(* IEC 61131-3 sources: 2026_Projet_YGO_ExcavatriceDragage/TOOLS/TEST_AUTO_CI/RESULTS/_TROUBLESHOOTING/tests, 5 files *)

(* ---- test_arb_cmd_both_atomic.st ---- *)
(* =========================================================================
   TEST CI AD HOC - Atomicite commande Both M1/M2 (T216, criticite C4)
   -------------------------------------------------------------------------
   Prouve les invariants de securite du depart couple des treuils M1/M2 :
     #1  Atomicite Both descente : BothDescendPermit=FALSE (un permit M2 absent)
         -> AUCUN des deux treuils ne demarre (StartStop M1=FALSE ET M2=FALSE).
     #2  Both nominal montee : les 2 permits agreges OK -> les DEUX demarrent.
     #3  Preservation unitaire : M1 seul / M2 seul / action benne M2 -> le gate
         Both*Permit est inactif, comportement inchange (aucun blocage croise).
     #4  Soft-stop : Both + ecart mineur -> jamais de demarrage unilateral (les 2
         bloques ensemble si le permit Both manque) ; hors Both (unitaire), l'ecart
         mineur bloque toujours le sens concerne (comportement preserve).
   Noms figes T216 intacts : EffectivePermitM1/2_Ascent/Descend non re-nommes.
   Chaque appel arb1(...)/arb2(...) = 1 scan de l'arbitre.
   (Le gate sync mineur de PRG_04 est coupe en Both en amont - voir le FB - ici on
   prouve que l'arbitre ne part JAMAIS seul, quelle que soit la polarite du flag.)
   ========================================================================= *)

SETUP
VAR
    arb1 : FB_WinchCmdArbitrationM1;
    arb2 : FB_WinchCmdArbitrationM2;
    joy  : ST_AcquisitionJoystickQualified;
    auth : ST_Modes_Autorisations;
    req  : ST_ProgramWinchRequest;
    both : ST_WinchBothIntent;
    ihm  : ST_fbWinchCmdArbitration_IHM;
    ctx  : ST_fbWinchCmdArbitration_Context;
    cfg1 : ST_fbWinchCmdArbitration_Cfg;
    cfg2 : ST_fbWinchCmdArbitration_Cfg;
END_VAR
END_SETUP

TEST 'T216 #1 Atomicite Both descente : BothDescendPermit=FALSE -> AUCUN treuil ne demarre'
    // Contexte : mode manuel boutons, intention both descente active.
    auth.Mode := E_Mode.MAINT_N1;
    auth.JoystickWinchSelectArbitrated := 0;
    both.Active := TRUE; both.Direction := -1;
    // Simule EffectivePermitM2_Descend=FALSE -> BothDescendPermit=FALSE (agregat PRG_04).
    ctx.BothDescendPermit := FALSE; ctx.BothAscentPermit := TRUE;
    ctx.BothBlock := TRUE;
    ctx.BucketBusy := FALSE; ctx.WinchBothMotionBlockedByBucket := FALSE;
    ctx.SyncBlocksAscent := FALSE; ctx.SyncBlocksDescent := FALSE;
    ihm.BtnAscentM1 := FALSE; ihm.BtnDescentM1 := FALSE;
    ihm.BtnAscentM2 := FALSE; ihm.BtnDescentM2 := FALSE;
    cfg1.BtnStepTgt := 5; cfg2.BtnStepTgt := 5; cfg2.BucketOverrideStepTgt := 1;

    arb1(Enable := TRUE, Joystick := joy, Auth := auth, ReqWinch := req,
         BothIntent := both, IHM := ihm, TglJoystickMaster := FALSE,
         Context := ctx, Cfg := cfg1);
    arb2(Enable := TRUE, Joystick := joy, Auth := auth, ReqWinch := req,
         BothIntent := both, IHM := ihm, TglJoystickMaster := FALSE,
         Context := ctx, Cfg := cfg2);

    ASSERT_FALSE(arb1.StartStop, 'T216#1 Both descente : StartStop M1=FALSE (permit Both manquant)');
    ASSERT_FALSE(arb2.StartStop, 'T216#1 Both descente : StartStop M2=FALSE (permit Both manquant)');
    ASSERT_EQ(arb1.Direction, -1, 'T216#1 l intention descente est portee, seule la commande est coupee');
END_TEST

TEST 'T216 #2 Both nomiinal montee : permits OK -> les DEUX demarrent ensemble'
    auth.Mode := E_Mode.MAINT_N1;
    auth.JoystickWinchSelectArbitrated := 0;
    both.Active := TRUE; both.Direction := 1;
    ctx.BothDescendPermit := TRUE; ctx.BothAscentPermit := TRUE;
    ctx.BothBlock := FALSE;
    ctx.BucketBusy := FALSE; ctx.WinchBothMotionBlockedByBucket := FALSE;
    ctx.SyncBlocksAscent := FALSE; ctx.SyncBlocksDescent := FALSE;
    ihm.BtnAscentM1 := FALSE; ihm.BtnDescentM1 := FALSE;
    ihm.BtnAscentM2 := FALSE; ihm.BtnDescentM2 := FALSE;
    cfg1.BtnStepTgt := 5; cfg2.BtnStepTgt := 5; cfg2.BucketOverrideStepTgt := 1;

    arb1(Enable := TRUE, Joystick := joy, Auth := auth, ReqWinch := req,
         BothIntent := both, IHM := ihm, TglJoystickMaster := FALSE,
         Context := ctx, Cfg := cfg1);
    arb2(Enable := TRUE, Joystick := joy, Auth := auth, ReqWinch := req,
         BothIntent := both, IHM := ihm, TglJoystickMaster := FALSE,
         Context := ctx, Cfg := cfg2);

    ASSERT_TRUE(arb1.StartStop, 'T216#2 Both montee : M1 demarre (permit OK)');
    ASSERT_TRUE(arb2.StartStop, 'T216#2 Both montee : M2 demarre (permit OK)');
    ASSERT_EQ(arb1.Direction, 1, 'T216#2 M1 sens montee');
    ASSERT_EQ(arb2.Direction, 1, 'T216#2 M2 sens montee');
END_TEST

TEST 'T216 #3a M1 seul : gate Both inactif (pas de blocage croise)'
    auth.Mode := E_Mode.MAINT_N1;
    auth.JoystickWinchSelectArbitrated := 1;
    both.Active := FALSE; both.Direction := 0;
    // Meme si les permits Both sont faux, le pilotage unitaire M1 n'en depend pas.
    ctx.BothDescendPermit := FALSE; ctx.BothAscentPermit := FALSE;
    ctx.BothBlock := FALSE;
    ctx.BucketBusy := FALSE; ctx.WinchBothMotionBlockedByBucket := FALSE;
    ctx.SyncBlocksAscent := FALSE; ctx.SyncBlocksDescent := FALSE;
    ihm.BtnAscentM1 := TRUE; ihm.BtnDescentM1 := FALSE;
    cfg1.BtnStepTgt := 5; cfg2.BtnStepTgt := 5; cfg2.BucketOverrideStepTgt := 1;

    arb1(Enable := TRUE, Joystick := joy, Auth := auth, ReqWinch := req,
         BothIntent := both, IHM := ihm, TglJoystickMaster := FALSE,
         Context := ctx, Cfg := cfg1);

    ASSERT_TRUE(arb1.StartStop, 'T216#3a M1 seul : demarre (couplage Both inactif)');
    ASSERT_EQ(arb1.Direction, 1, 'T216#3a M1 sens montee');
END_TEST

TEST 'T216 #3b M2 seul : gate Both inactif (pas de blocage croise)'
    auth.Mode := E_Mode.MAINT_N1;
    auth.JoystickWinchSelectArbitrated := 2;
    both.Active := FALSE; both.Direction := 0;
    ctx.BothDescendPermit := FALSE; ctx.BothAscentPermit := FALSE;
    ctx.BothBlock := FALSE;
    ctx.BucketBusy := FALSE; ctx.WinchBothMotionBlockedByBucket := FALSE;
    ctx.SyncBlocksAscent := FALSE; ctx.SyncBlocksDescent := FALSE;
    ihm.BtnAscentM2 := TRUE;

    arb2(Enable := TRUE, Joystick := joy, Auth := auth, ReqWinch := req,
         BothIntent := both, IHM := ihm, TglJoystickMaster := FALSE,
         Context := ctx, Cfg := cfg2);

    ASSERT_TRUE(arb2.StartStop, 'T216#3b M2 seul : demarre (couplage Both inactif)');
    ASSERT_EQ(arb2.Direction, 1, 'T216#3b M2 sens montee');
END_TEST

TEST 'T216 #3c benne M2 : chemin override preserve (hors gate Both)'
    auth.Mode := E_Mode.MAINT_N1;
    both.Active := FALSE; both.Direction := 0;
    ctx.BothDescendPermit := FALSE; ctx.BothAscentPermit := FALSE;
    ctx.BothBlock := FALSE;
    // Action benne M2 active (chemin override FB_WinchCmdArbitrationM2).
    ctx.BucketBusy := TRUE; ctx.BucketM2StartStop := TRUE; ctx.BucketM2Open := TRUE;
    ctx.WinchBothMotionBlockedByBucket := FALSE;
    ctx.SyncBlocksAscent := FALSE; ctx.SyncBlocksDescent := FALSE;
    cfg2.BucketOverrideStepTgt := 1;

    arb2(Enable := TRUE, Joystick := joy, Auth := auth, ReqWinch := req,
         BothIntent := both, IHM := ihm, TglJoystickMaster := FALSE,
         Context := ctx, Cfg := cfg2);

    ASSERT_TRUE(arb2.StartStop, 'T216#3c action benne M2 : demarre (override hors gate Both)');
    ASSERT_EQ(arb2.StepTgt, 1, 'T216#3c action benne M2 : palier lent override');
END_TEST

TEST 'T216 #4a Both + ecart mineur : JAMAIS de demarrage unilateral (les DEUX bloques)'
    auth.Mode := E_Mode.MAINT_N1;
    auth.JoystickWinchSelectArbitrated := 0;
    both.Active := TRUE; both.Direction := -1;
    ctx.BothDescendPermit := FALSE;   // un permit Both manquant (M2)
    ctx.BothAscentPermit := TRUE;
    ctx.BothBlock := TRUE;
    ctx.BucketBusy := FALSE; ctx.WinchBothMotionBlockedByBucket := FALSE;
    // M1 bloque sur SyncBlocksAscent ; en descente M2 bloque sur SyncBlocksDescent.
    // Quelle que soit la polarite, le gate Both (permit manquant) bloque les DEUX.
    ctx.SyncBlocksAscent := TRUE; ctx.SyncBlocksDescent := TRUE;

    arb1(Enable := TRUE, Joystick := joy, Auth := auth, ReqWinch := req,
         BothIntent := both, IHM := ihm, TglJoystickMaster := FALSE,
         Context := ctx, Cfg := cfg1);
    arb2(Enable := TRUE, Joystick := joy, Auth := auth, ReqWinch := req,
         BothIntent := both, IHM := ihm, TglJoystickMaster := FALSE,
         Context := ctx, Cfg := cfg2);

    ASSERT_FALSE(arb1.StartStop, 'T216#4a Both + ecart : M1 bloque (pas de depart unilateral)');
    ASSERT_FALSE(arb2.StartStop, 'T216#4a Both + ecart : M2 bloque (pas de depart unilateral)');
END_TEST

TEST 'T216 #4b unite + ecart mineur : le sens concerne reste bloque (preservation)'
    auth.Mode := E_Mode.MAINT_N1;
    auth.JoystickWinchSelectArbitrated := 1;
    both.Active := FALSE; both.Direction := 0;
    ctx.BothDescendPermit := FALSE; ctx.BothAscentPermit := FALSE;
    ctx.BothBlock := FALSE;
    ctx.BucketBusy := FALSE; ctx.WinchBothMotionBlockedByBucket := FALSE;
    // Montee M1 bloquee par l'ecart mineur si SyncBlocksAscent (comportement d'origine
    // hors Both, preserve).
    ctx.SyncBlocksAscent := TRUE; ctx.SyncBlocksDescent := FALSE;
    ihm.BtnAscentM1 := TRUE;

    arb1(Enable := TRUE, Joystick := joy, Auth := auth, ReqWinch := req,
         BothIntent := both, IHM := ihm, TglJoystickMaster := FALSE,
         Context := ctx, Cfg := cfg1);

    ASSERT_FALSE(arb1.StartStop, 'T216#4b M1 seul + ecart mineur montee : bloque (comportement preserve hors Both)');
END_TEST

(* ---- test_fb_encoder_speedmeasure.st ---- *)
SETUP
VAR
    fb : FB_Encoder_SpeedMeasure;
END_VAR
END_SETUP

TEST 'TC-T084-001 Mesure dynamique 1.0 m/s et 2.0 m/s sur fenetre glissante 50ms'
    (* Scan 0 : Neutralisation initiale *)
    fb(Enable := FALSE, Reset := FALSE, Position_M := 0.0, PositionValid := FALSE);
    ASSERT_FALSE(fb.Valid, 'Enable=FALSE -> Valid=FALSE');
    ASSERT_EQ(fb.Speed_Mps, 0.0, 'Enable=FALSE -> Speed=0');

    ADVANCE_TIME(10000000); (* +10 ms *)

    (* Scan 1 (t=10ms) : Activation et premier echantillon a 0.0 m *)
    fb(Enable := TRUE, Reset := FALSE, Position_M := 0.0, PositionValid := TRUE);
    ASSERT_FALSE(fb.Valid, 'Echantillon 1 : Fenetre 50ms pas encore remplie');

    ADVANCE_TIME(10000000); (* +10 ms (t=20ms) *)

    (* Scan 2 (t=20ms) : Deplacement a v=1.0 m/s -> pos = 0.01 m (+10mm en 10ms) *)
    fb(Enable := TRUE, Reset := FALSE, Position_M := 0.01, PositionValid := TRUE);
    ASSERT_FALSE(fb.Valid, 'Echantillon 2 : Fenetre 50ms pas encore remplie');

    ADVANCE_TIME(10000000); (* +10 ms (t=30ms) *)

    (* Scan 3 (t=30ms) : pos = 0.02 m *)
    fb(Enable := TRUE, Reset := FALSE, Position_M := 0.02, PositionValid := TRUE);
    ASSERT_FALSE(fb.Valid, 'Echantillon 3 : Fenetre 50ms pas encore remplie');

    ADVANCE_TIME(10000000); (* +10 ms (t=40ms) *)

    (* Scan 4 (t=40ms) : pos = 0.03 m *)
    fb(Enable := TRUE, Reset := FALSE, Position_M := 0.03, PositionValid := TRUE);
    ASSERT_FALSE(fb.Valid, 'Echantillon 4 : Fenetre 50ms pas encore remplie');

    ADVANCE_TIME(10000000); (* +10 ms (t=50ms) *)

    (* Scan 5 (t=50ms) : pos = 0.04 m *)
    fb(Enable := TRUE, Reset := FALSE, Position_M := 0.04, PositionValid := TRUE);
    ASSERT_FALSE(fb.Valid, 'Echantillon 5 : Fenetre 50ms pas encore remplie');

    ADVANCE_TIME(10000000); (* +10 ms (t=60ms) *)

    (* Scan 6 (t=60ms) : pos = 0.05 m -> 6 echantillons couvrant 50ms (t=10ms a t=60ms) *)
    fb(Enable := TRUE, Reset := FALSE, Position_M := 0.05, PositionValid := TRUE);
    ASSERT_TRUE(fb.Valid, '6 echantillons sur 50ms atteints -> Valid=TRUE');
    ASSERT_NEAR(fb.Speed_Mps, 1.0, 0.05, 'Vitesse absolue mesuree = 1.0 m/s');
    ASSERT_NEAR(fb.SignedSpeed_Mps, 1.0, 0.05, 'Vitesse signee montee = +1.0 m/s');

    ADVANCE_TIME(10000000); (* +10 ms (t=70ms) *)

    (* Scan 7 (t=70ms) : Acceleration a 2.0 m/s (+20mm en 10ms) -> pos = 0.07 m *)
    fb(Enable := TRUE, Reset := FALSE, Position_M := 0.07, PositionValid := TRUE);
    ASSERT_TRUE(fb.Valid, 'Fenetre glissante active');
    ASSERT_NEAR(fb.Speed_Mps, 1.2, 0.05, 'Transition glissante vers 2.0 m/s (pos 0.07 - pos 0.01 = 0.06m / 50ms = 1.2 m/s)');

    ADVANCE_TIME(10000000); (* +10 ms (t=80ms) *)

    (* Scan 8 (t=80ms) : Suite a 2.0 m/s -> pos = 0.09 m *)
    fb(Enable := TRUE, Reset := FALSE, Position_M := 0.09, PositionValid := TRUE);
    ASSERT_TRUE(fb.Valid, 'Fenetre glissante active');
    ASSERT_NEAR(fb.Speed_Mps, 1.4, 0.05, 'Transition glissante vers 2.0 m/s (pos 0.09 - pos 0.02 = 0.07m / 50ms = 1.4 m/s)');

    ADVANCE_TIME(10000000); (* +10 ms (t=90ms) *)

    (* Scan 9 (t=90ms) : Descente a -2.0 m/s (-20mm en 10ms) -> pos = 0.07 m *)
    fb(Enable := TRUE, Reset := FALSE, Position_M := 0.07, PositionValid := TRUE);
    ASSERT_TRUE(fb.Valid, 'Fenetre glissante active');

    ADVANCE_TIME(10000000); (* +10 ms (t=100ms) *)

    (* Scan 10 (t=100ms) : Coupure PositionValid=FALSE -> Purge immediate *)
    fb(Enable := TRUE, Reset := FALSE, Position_M := 0.07, PositionValid := FALSE);
    ASSERT_FALSE(fb.Valid, 'Rupture confiance PositionValid=FALSE -> Valid retombe immediatement a FALSE');
    ASSERT_EQ(fb.Speed_Mps, 0.0, 'Purge immediate -> Speed=0.0');
    ASSERT_EQ(fb.SignedSpeed_Mps, 0.0, 'Purge immediate -> SignedSpeed=0.0');
END_TEST

(* ---- test_fb_sim_joystick.st ---- *)
(* ═══════════════════════════════════════════════════════════════════════
   🕵️ TEST CI AD HOC — FB_Joystick / ArmingPermit (LOT_JOYSTICK_ARMINGPERMIT)
   ───────────────────────────────────────────────────────────────────────
   Prouve les critères d'acceptation AC1/AC2/AC3 du contrat
   TASK_CONTRACT_JOYSTICK_ARMINGPERMIT.yaml :
     • AC1 : ArmingPermit=FALSE + appui 110ms -> DeadmanArmed=FALSE ;
             ArmingPermit=TRUE  + appui 110ms -> DeadmanArmed=TRUE.
     • AC2 : ArmingPermit=FALSE -> AxisCmdX/Y.Enable=FALSE, SpeedRef=0,
             warning "armement non permis" actif (sortie ArmingPermitDenied).
     • AC3 : RawOutOfRange=TRUE -> Enable=FALSE même si ArmingPermit=TRUE ;
             ArmingPermit=FALSE bloque l'armement même sans défaut capteur.
   ⚠️ Chaque appel fb(...) = 1 scan (10ms) ; ADVANCE_TIME avance le temps simulé
   sans faire tourner le FB. Un maintien de 110ms = front + ADVANCE_TIME + rappel.
   ⚠️ STruCpp ne re-copie PAS la sortie VAR_IN_OUT (NeutralXMem/YMem) entre deux
   appels -> nx/ny ré-injectés avant chaque appel (limite outillage documentée).
   Chaque TEST remet l'état armement à zéro via un premier appel ENABLE:=FALSE
   (le gate remet DeadmanArmed/DeadmanArmPending/ArmingPermitDenied/timers) pour
   être autonome quelle que soit l'instance FB.
   ═══════════════════════════════════════════════════════════════════════ *)

SETUP
VAR
    fb : FB_JOYSTICK;
    nx : INT := 5000;
    ny : INT := 5000;
    diagOk : ST_DIAG_DEVICE;
END_VAR
END_SETUP

TEST 'AC1a : ArmingPermit=FALSE bloque l armement (appui maintenu 110ms)'
    diagOk.ONLINE := TRUE; diagOk.OPERATIONAL := TRUE; diagOk.ERROR := FALSE;
    diagOk.ERRORID := 0; diagOk.STATE := E_DIAG_STATE.READY; diagOk.STATEATERROR := E_DIAG_STATE.DISABLED;
    nx := 5000; ny := 5000;

    (* reset etat armement via le gate Enable=FALSE *)
    fb(ENABLE := FALSE, RESET := FALSE,
       ARMINGPERMIT := FALSE,
       BUSCANOPENOP := diagOk, JOYSTICKOP := diagOk,
       RAWX := 5000, RAWY := 5000, RAWBUTTON := FALSE, BTNCALIBRATE := FALSE,
       INVERTX := FALSE, INVERTY := FALSE, DEADBANDRAW := 300,
       NEUTRALHOLDTIME := T#100MS, DEADMANARMHOLDTIME := T#100MS, DEADMANARMGRACETIME := T#3S,
       NEUTRALXMEM := nx, NEUTRALYMEM := ny);

    (* front appui, ArmingPermit=FALSE : la permission refuse le démarrage du timer
       d'armement -> DeadmanArmed ne doit JAMAIS passer à TRUE. *)
    fb(ENABLE := TRUE, RESET := FALSE,
       ARMINGPERMIT := FALSE,
       BUSCANOPENOP := diagOk, JOYSTICKOP := diagOk,
       RAWX := 5000, RAWY := 5000, RAWBUTTON := TRUE, BTNCALIBRATE := FALSE,
       INVERTX := FALSE, INVERTY := FALSE, DEADBANDRAW := 300,
       NEUTRALHOLDTIME := T#100MS, DEADMANARMHOLDTIME := T#100MS, DEADMANARMGRACETIME := T#3S,
       NEUTRALXMEM := nx, NEUTRALYMEM := ny);
    ADVANCE_TIME(110000000);   (* maintien 110ms >= DeadmanArmHoldTime 100ms *)
    fb(ENABLE := TRUE, RESET := FALSE,
       ARMINGPERMIT := FALSE,
       BUSCANOPENOP := diagOk, JOYSTICKOP := diagOk,
       RAWX := 5000, RAWY := 5000, RAWBUTTON := TRUE, BTNCALIBRATE := FALSE,
       INVERTX := FALSE, INVERTY := FALSE, DEADBANDRAW := 300,
       NEUTRALHOLDTIME := T#100MS, DEADMANARMHOLDTIME := T#100MS, DEADMANARMGRACETIME := T#3S,
       NEUTRALXMEM := nx, NEUTRALYMEM := ny);
    ASSERT_FALSE(fb.DEADMANARMED, 'AC1 : ArmingPermit=FALSE + appui 110ms -> DeadmanArmed reste FALSE (armement bloque)');
END_TEST

TEST 'AC1b : ArmingPermit=TRUE autorise l armement (appui maintenu 110ms)'
    diagOk.ONLINE := TRUE; diagOk.OPERATIONAL := TRUE; diagOk.ERROR := FALSE;
    diagOk.ERRORID := 0; diagOk.STATE := E_DIAG_STATE.READY; diagOk.STATEATERROR := E_DIAG_STATE.DISABLED;
    nx := 5000; ny := 5000;

    fb(ENABLE := FALSE, RESET := FALSE,
       ARMINGPERMIT := TRUE,
       BUSCANOPENOP := diagOk, JOYSTICKOP := diagOk,
       RAWX := 5000, RAWY := 5000, RAWBUTTON := FALSE, BTNCALIBRATE := FALSE,
       INVERTX := FALSE, INVERTY := FALSE, DEADBANDRAW := 300,
       NEUTRALHOLDTIME := T#100MS, DEADMANARMHOLDTIME := T#100MS, DEADMANARMGRACETIME := T#3S,
       NEUTRALXMEM := nx, NEUTRALYMEM := ny);

    (* front appui, ArmingPermit=TRUE : maintien complet -> armement normal *)
    fb(ENABLE := TRUE, RESET := FALSE,
       ARMINGPERMIT := TRUE,
       BUSCANOPENOP := diagOk, JOYSTICKOP := diagOk,
       RAWX := 5000, RAWY := 5000, RAWBUTTON := TRUE, BTNCALIBRATE := FALSE,
       INVERTX := FALSE, INVERTY := FALSE, DEADBANDRAW := 300,
       NEUTRALHOLDTIME := T#100MS, DEADMANARMHOLDTIME := T#100MS, DEADMANARMGRACETIME := T#3S,
       NEUTRALXMEM := nx, NEUTRALYMEM := ny);
    ADVANCE_TIME(110000000);   (* maintien 110ms >= DeadmanArmHoldTime 100ms *)
    fb(ENABLE := TRUE, RESET := FALSE,
       ARMINGPERMIT := TRUE,
       BUSCANOPENOP := diagOk, JOYSTICKOP := diagOk,
       RAWX := 5000, RAWY := 5000, RAWBUTTON := TRUE, BTNCALIBRATE := FALSE,
       INVERTX := FALSE, INVERTY := FALSE, DEADBANDRAW := 300,
       NEUTRALHOLDTIME := T#100MS, DEADMANARMHOLDTIME := T#100MS, DEADMANARMGRACETIME := T#3S,
       NEUTRALXMEM := nx, NEUTRALYMEM := ny);
    ASSERT_TRUE(fb.DEADMANARMED, 'AC1 : ArmingPermit=TRUE + appui 110ms -> DeadmanArmed=TRUE (armement autorise)');
END_TEST

TEST 'AC2 : ArmingPermit=FALSE -> Enable=FALSE, SpeedRef=0, warning armement non permis actif'
    diagOk.ONLINE := TRUE; diagOk.OPERATIONAL := TRUE; diagOk.ERROR := FALSE;
    diagOk.ERRORID := 0; diagOk.STATE := E_DIAG_STATE.READY; diagOk.STATEATERROR := E_DIAG_STATE.DISABLED;
    nx := 5000; ny := 5000;

    fb(ENABLE := FALSE, RESET := FALSE,
       ARMINGPERMIT := FALSE,
       BUSCANOPENOP := diagOk, JOYSTICKOP := diagOk,
       RAWX := 5000, RAWY := 5000, RAWBUTTON := FALSE, BTNCALIBRATE := FALSE,
       INVERTX := FALSE, INVERTY := FALSE, DEADBANDRAW := 300,
       NEUTRALHOLDTIME := T#100MS, DEADMANARMHOLDTIME := T#100MS, DEADMANARMGRACETIME := T#3S,
       NEUTRALXMEM := nx, NEUTRALYMEM := ny);

    (* appui maintenu, ArmingPermit=FALSE : armement bloqué. On pousse même l'axe X/Y
       (RawX/Y=8000) pour prouver qu'AUCUNE commande de mouvement n'est émise. *)
    fb(ENABLE := TRUE, RESET := FALSE,
       ARMINGPERMIT := FALSE,
       BUSCANOPENOP := diagOk, JOYSTICKOP := diagOk,
       RAWX := 5000, RAWY := 5000, RAWBUTTON := TRUE, BTNCALIBRATE := FALSE,
       INVERTX := FALSE, INVERTY := FALSE, DEADBANDRAW := 300,
       NEUTRALHOLDTIME := T#100MS, DEADMANARMHOLDTIME := T#100MS, DEADMANARMGRACETIME := T#3S,
       NEUTRALXMEM := nx, NEUTRALYMEM := ny);
    ADVANCE_TIME(110000000);
    fb(ENABLE := TRUE, RESET := FALSE,
       ARMINGPERMIT := FALSE,
       BUSCANOPENOP := diagOk, JOYSTICKOP := diagOk,
       RAWX := 8000, RAWY := 8000, RAWBUTTON := TRUE, BTNCALIBRATE := FALSE,
       INVERTX := FALSE, INVERTY := FALSE, DEADBANDRAW := 300,
       NEUTRALHOLDTIME := T#100MS, DEADMANARMHOLDTIME := T#100MS, DEADMANARMGRACETIME := T#3S,
       NEUTRALXMEM := nx, NEUTRALYMEM := ny);
    ASSERT_FALSE(fb.DEADMANARMED, 'AC2 : pre-requis - armement bloque (jamais arme)');
    ASSERT_FALSE(fb.AXISCMDX.ENABLE, 'AC2 : ArmingPermit=FALSE -> AxisCmdX.Enable=FALSE (pipeline neutralise)');
    ASSERT_FALSE(fb.AXISCMDY.ENABLE, 'AC2 : ArmingPermit=FALSE -> AxisCmdY.Enable=FALSE');
    ASSERT_NEAR(fb.AXISCMDX.SPEEDREF, 0.0, 0.01, 'AC2 : SpeedRef axe X = 0 (aucune commande de mouvement)');
    ASSERT_NEAR(fb.AXISCMDY.SPEEDREF, 0.0, 0.01, 'AC2 : SpeedRef axe Y = 0');
    ASSERT_TRUE(fb.ARMINGPERMITDENIED, 'AC2 : warning "armement non permis" actif (sortie dediee ArmingPermitDenied)');
END_TEST

TEST 'AC3a : defaut capteur (RawOutOfRange) neutralise Enable meme si ArmingPermit=TRUE'
    diagOk.ONLINE := TRUE; diagOk.OPERATIONAL := TRUE; diagOk.ERROR := FALSE;
    diagOk.ERRORID := 0; diagOk.STATE := E_DIAG_STATE.READY; diagOk.STATEATERROR := E_DIAG_STATE.DISABLED;
    nx := 5000; ny := 5000;

    fb(ENABLE := FALSE, RESET := FALSE,
       ARMINGPERMIT := TRUE,
       BUSCANOPENOP := diagOk, JOYSTICKOP := diagOk,
       RAWX := 5000, RAWY := 5000, RAWBUTTON := FALSE, BTNCALIBRATE := FALSE,
       INVERTX := FALSE, INVERTY := FALSE, DEADBANDRAW := 300,
       NEUTRALHOLDTIME := T#100MS, DEADMANARMHOLDTIME := T#100MS, DEADMANARMGRACETIME := T#3S,
       NEUTRALXMEM := nx, NEUTRALYMEM := ny);

    (* arme d'abord avec ArmingPermit=TRUE *)
    fb(ENABLE := TRUE, RESET := FALSE,
       ARMINGPERMIT := TRUE,
       BUSCANOPENOP := diagOk, JOYSTICKOP := diagOk,
       RAWX := 5000, RAWY := 5000, RAWBUTTON := TRUE, BTNCALIBRATE := FALSE,
       INVERTX := FALSE, INVERTY := FALSE, DEADBANDRAW := 300,
       NEUTRALHOLDTIME := T#100MS, DEADMANARMHOLDTIME := T#100MS, DEADMANARMGRACETIME := T#3S,
       NEUTRALXMEM := nx, NEUTRALYMEM := ny);
    ADVANCE_TIME(110000000);
    fb(ENABLE := TRUE, RESET := FALSE,
       ARMINGPERMIT := TRUE,
       BUSCANOPENOP := diagOk, JOYSTICKOP := diagOk,
       RAWX := 5000, RAWY := 5000, RAWBUTTON := TRUE, BTNCALIBRATE := FALSE,
       INVERTX := FALSE, INVERTY := FALSE, DEADBANDRAW := 300,
       NEUTRALHOLDTIME := T#100MS, DEADMANARMHOLDTIME := T#100MS, DEADMANARMGRACETIME := T#3S,
       NEUTRALXMEM := nx, NEUTRALYMEM := ny);
    ASSERT_TRUE(fb.DEADMANARMED, 'AC3a : pre-requis - geste arme avec ArmingPermit=TRUE');

    (* défaut capteur (RawX/RawY hors plage ADC + marge) : Enable doit tomber à FALSE,
       indépendamment d'ArmingPermit (mécanisme interne de perte de confiance) *)
    ADVANCE_TIME(10000000);
    fb(ENABLE := TRUE, RESET := FALSE,
       ARMINGPERMIT := TRUE,
       BUSCANOPENOP := diagOk, JOYSTICKOP := diagOk,
       RAWX := 20000, RAWY := 20000, RAWBUTTON := TRUE, BTNCALIBRATE := FALSE,
       INVERTX := FALSE, INVERTY := FALSE, DEADBANDRAW := 300,
       NEUTRALHOLDTIME := T#100MS, DEADMANARMHOLDTIME := T#100MS, DEADMANARMGRACETIME := T#3S,
       NEUTRALXMEM := nx, NEUTRALYMEM := ny);
    ASSERT_FALSE(fb.AXISCMDX.ENABLE, 'AC3a : RawOutOfRange=TRUE -> AxisCmdX.Enable=FALSE meme si ArmingPermit=TRUE');
    ASSERT_FALSE(fb.AXISCMDY.ENABLE, 'AC3a : meme comportement axe Y');
    ASSERT_NEAR(fb.AXISCMDX.SPEEDREF, 0.0, 0.01, 'AC3a : SpeedRef X coupee sur defaut capteur');
    ASSERT_NEAR(fb.AXISCMDY.SPEEDREF, 0.0, 0.01, 'AC3a : SpeedRef Y coupee');
END_TEST

TEST 'AC3b : ArmingPermit=FALSE bloque l armement meme sans defaut capteur'
    diagOk.ONLINE := TRUE; diagOk.OPERATIONAL := TRUE; diagOk.ERROR := FALSE;
    diagOk.ERRORID := 0; diagOk.STATE := E_DIAG_STATE.READY; diagOk.STATEATERROR := E_DIAG_STATE.DISABLED;
    nx := 5000; ny := 5000;

    fb(ENABLE := FALSE, RESET := FALSE,
       ARMINGPERMIT := FALSE,
       BUSCANOPENOP := diagOk, JOYSTICKOP := diagOk,
       RAWX := 5000, RAWY := 5000, RAWBUTTON := FALSE, BTNCALIBRATE := FALSE,
       INVERTX := FALSE, INVERTY := FALSE, DEADBANDRAW := 300,
       NEUTRALHOLDTIME := T#100MS, DEADMANARMHOLDTIME := T#100MS, DEADMANARMGRACETIME := T#3S,
       NEUTRALXMEM := nx, NEUTRALYMEM := ny);

    (* capteur SAIN (RawX/RawY = 5000, dans plage) + ArmingPermit=FALSE : malgré un appui
       maintenu 110ms, l'armement reste bloqué (la permission, pas un défaut capteur). *)
    fb(ENABLE := TRUE, RESET := FALSE,
       ARMINGPERMIT := FALSE,
       BUSCANOPENOP := diagOk, JOYSTICKOP := diagOk,
       RAWX := 5000, RAWY := 5000, RAWBUTTON := TRUE, BTNCALIBRATE := FALSE,
       INVERTX := FALSE, INVERTY := FALSE, DEADBANDRAW := 300,
       NEUTRALHOLDTIME := T#100MS, DEADMANARMHOLDTIME := T#100MS, DEADMANARMGRACETIME := T#3S,
       NEUTRALXMEM := nx, NEUTRALYMEM := ny);
    ADVANCE_TIME(110000000);
    fb(ENABLE := TRUE, RESET := FALSE,
       ARMINGPERMIT := FALSE,
       BUSCANOPENOP := diagOk, JOYSTICKOP := diagOk,
       RAWX := 5000, RAWY := 5000, RAWBUTTON := TRUE, BTNCALIBRATE := FALSE,
       INVERTX := FALSE, INVERTY := FALSE, DEADBANDRAW := 300,
       NEUTRALHOLDTIME := T#100MS, DEADMANARMHOLDTIME := T#100MS, DEADMANARMGRACETIME := T#3S,
       NEUTRALXMEM := nx, NEUTRALYMEM := ny);
    ASSERT_FALSE(fb.DEADMANARMED, 'AC3b : ArmingPermit=FALSE bloque l armement meme sans defaut capteur');
    ASSERT_EQ(fb.ERRORID, 0, 'AC3b : capteur sain -> aucun defaut capteur leve (blocage purement par permission)');
END_TEST

(* ---- test_fb_winch_minstepdown.st ---- *)
(* =======================================================================
   🧪 test ad hoc troubleshooting — FB_Winch / plancher MinStepDown
   Sujet : TROUBLESHOOTING_TreuilM2_LimiteDescente_20260901
   Symptôme : DescendPermit=FALSE (limite basse atteinte) mais descente
   continue au palier 1 jusqu'à -20 m. Reproduit le snapshot 01:48 :
   Direction=-1, StartStop=TRUE, MinStepDown=1 (CommonMinStepDown=MAX(1,·)).
   Question tranchée : le plancher MinStepDown relève-t-il RequestedStep
   à >= 1 APRÈS que EffectiveSafeStop (permis descente refusé) a mis la
   cible à 0 ? ATTENDU CORRECT : StepNumber=0, RelayRev=FALSE.
   ======================================================================= *)

SETUP
VAR
    FB_W : FB_Winch;
    Table : ST_SpeedStepTable;
    DriveReq : ST_fbWinch_DriveRequest;
    Sens : ST_fbWinch_Sensors;
    Cfg : ST_fbWinch_Cfg;
END_VAR
END_SETUP

TEST 'TROUBLESHOOT-01 Descente permise : MinStepDown=1 -> palier 1 maintenu (comportement nominal plongee)'
    Table.StepThreshold_Pct[1] := 10.0;
    Table.StepThreshold_Pct[2] := 30.0;
    Table.StepThreshold_Pct[3] := 50.0;
    Table.StepThreshold_Pct[4] := 70.0;
    Table.StepThreshold_Pct[5] := 90.0;
    Table.P2R1 := TRUE;
    Table.P3R1 := TRUE;
    Table.P4R1 := TRUE;
    Table.P5R1 := TRUE;
    Cfg.SpeedStepTable := Table;
    Sens.Homed := TRUE;
    Sens.ContactorsAllOff := TRUE;
    Sens.SpeedGuardReady := TRUE;

    // Scan 0 : regime nominal au NEUTRE (arme l interlock direction)
    DriveReq.StartStop := FALSE;
    DriveReq.Direction := 0;
    DriveReq.SpeedStepReq := 0;
    DriveReq.MinStepDown := 1;
    DriveReq.MaxStepDown := 3;
    DriveReq.BottomLimitM := -20.0;
    FB_W(Enable := TRUE, Reset := FALSE, PowerContactorEngaged := TRUE,
         DriveRequest := DriveReq, Sensors := Sens, Config := Cfg,
         SafeStop := FALSE, DescendPermit := TRUE, AscentPermit := TRUE);
    ADVANCE_TIME(10000000);
    FB_W(Enable := TRUE, Reset := FALSE, PowerContactorEngaged := TRUE,
         DriveRequest := DriveReq, Sensors := Sens, Config := Cfg,
         SafeStop := FALSE, DescendPermit := TRUE, AscentPermit := TRUE);
    ADVANCE_TIME(10000000);

    // Neutre -> descente : IMMEDIAT (pas d inversion)
    DriveReq.StartStop := TRUE;
    DriveReq.Direction := -1;
    DriveReq.SpeedStepReq := 1;
    FB_W(Enable := TRUE, Reset := FALSE, PowerContactorEngaged := TRUE,
         DriveRequest := DriveReq, Sensors := Sens, Config := Cfg,
         SafeStop := FALSE, DescendPermit := TRUE, AscentPermit := TRUE);
    ASSERT_EQ(FB_W.CommandedDirection, -1, 'Neutre->descente : direction -1 immediat');

    // Regime etabli (cadence descente 500ms)
    ADVANCE_TIME(10000000);
    FB_W(Enable := TRUE, Reset := FALSE, PowerContactorEngaged := TRUE,
         DriveRequest := DriveReq, Sensors := Sens, Config := Cfg,
         SafeStop := FALSE, DescendPermit := TRUE, AscentPermit := TRUE);
    ADVANCE_TIME(10000000);
    FB_W(Enable := TRUE, Reset := FALSE, PowerContactorEngaged := TRUE,
         DriveRequest := DriveReq, Sensors := Sens, Config := Cfg,
         SafeStop := FALSE, DescendPermit := TRUE, AscentPermit := TRUE);

    ASSERT_TRUE(FB_W.RelayRev, 'Permis OK + MinStepDown=1 -> descente energisee (nominal)');
    ASSERT_EQ(FB_W.StepNumber, 1, 'Plancher MinStepDown=1 -> palier 1 (nominal plongee)');
END_TEST

TEST 'TROUBLESHOOT-02 BUG ? DescendPermit=FALSE + MinStepDown=1 : la descente doit S ARRETER (limite basse atteinte)'
    Table.StepThreshold_Pct[1] := 10.0;
    Table.StepThreshold_Pct[2] := 30.0;
    Table.StepThreshold_Pct[3] := 50.0;
    Table.StepThreshold_Pct[4] := 70.0;
    Table.StepThreshold_Pct[5] := 90.0;
    Table.P2R1 := TRUE;
    Table.P3R1 := TRUE;
    Table.P4R1 := TRUE;
    Table.P5R1 := TRUE;
    Cfg.SpeedStepTable := Table;
    Sens.Homed := TRUE;
    Sens.ContactorsAllOff := TRUE;
    Sens.SpeedGuardReady := TRUE;

    // Phase 0 : neutre (arme l interlock)
    DriveReq.StartStop := FALSE;
    DriveReq.Direction := 0;
    DriveReq.SpeedStepReq := 0;
    DriveReq.MinStepDown := 1;
    DriveReq.MaxStepDown := 3;
    DriveReq.BottomLimitM := -20.0;
    FB_W(Enable := TRUE, Reset := FALSE, PowerContactorEngaged := TRUE,
         DriveRequest := DriveReq, Sensors := Sens, Config := Cfg,
         SafeStop := FALSE, DescendPermit := TRUE, AscentPermit := TRUE);
    ADVANCE_TIME(10000000);
    FB_W(Enable := TRUE, Reset := FALSE, PowerContactorEngaged := TRUE,
         DriveRequest := DriveReq, Sensors := Sens, Config := Cfg,
         SafeStop := FALSE, DescendPermit := TRUE, AscentPermit := TRUE);
    ADVANCE_TIME(10000000);

    // Phase 1 : descente normale (permis OK) pour etablir la direction + palier
    DriveReq.StartStop := TRUE;
    DriveReq.Direction := -1;
    DriveReq.SpeedStepReq := 1;
    FB_W(Enable := TRUE, Reset := FALSE, PowerContactorEngaged := TRUE,
         DriveRequest := DriveReq, Sensors := Sens, Config := Cfg,
         SafeStop := FALSE, DescendPermit := TRUE, AscentPermit := TRUE);
    ADVANCE_TIME(10000000);
    FB_W(Enable := TRUE, Reset := FALSE, PowerContactorEngaged := TRUE,
         DriveRequest := DriveReq, Sensors := Sens, Config := Cfg,
         SafeStop := FALSE, DescendPermit := TRUE, AscentPermit := TRUE);
    ADVANCE_TIME(10000000);
    FB_W(Enable := TRUE, Reset := FALSE, PowerContactorEngaged := TRUE,
         DriveRequest := DriveReq, Sensors := Sens, Config := Cfg,
         SafeStop := FALSE, DescendPermit := TRUE, AscentPermit := TRUE);

    ASSERT_TRUE(FB_W.RelayRev, 'Pre-condition : descente etablie (permis OK)');

    // Phase 2 : LE PERMIS DESCENTE TOMBE (limite basse atteinte) — l operateur maintient
    // la demande (StartStop=TRUE, Dir=-1, MinStepDown=1 : exactement le snapshot 01:48)
    ADVANCE_TIME(10000000);
    FB_W(Enable := TRUE, Reset := FALSE, PowerContactorEngaged := TRUE,
         DriveRequest := DriveReq, Sensors := Sens, Config := Cfg,
         SafeStop := FALSE, DescendPermit := FALSE, AscentPermit := TRUE);
    ADVANCE_TIME(10000000);
    FB_W(Enable := TRUE, Reset := FALSE, PowerContactorEngaged := TRUE,
         DriveRequest := DriveReq, Sensors := Sens, Config := Cfg,
         SafeStop := FALSE, DescendPermit := FALSE, AscentPermit := TRUE);
    ADVANCE_TIME(10000000);
    FB_W(Enable := TRUE, Reset := FALSE, PowerContactorEngaged := TRUE,
         DriveRequest := DriveReq, Sensors := Sens, Config := Cfg,
         SafeStop := FALSE, DescendPermit := FALSE, AscentPermit := TRUE);
    ADVANCE_TIME(10000000);
    FB_W(Enable := TRUE, Reset := FALSE, PowerContactorEngaged := TRUE,
         DriveRequest := DriveReq, Sensors := Sens, Config := Cfg,
         SafeStop := FALSE, DescendPermit := FALSE, AscentPermit := TRUE);

    // VERDICT : si ces assertions echouent, le bug plancher est CONFIRME mechaniquement
    ASSERT_EQ(FB_W.StepNumber, 0, 'Permis descente FALSE -> StepNumber doit retomber a 0');
    ASSERT_FALSE(FB_W.RelayRev, 'Permis descente FALSE -> RelayRev doit retomber (arret descente)');
END_TEST

TEST 'TROUBLESHOOT-03 Controle : DescendPermit=FALSE SANS plancher (MinStepDown=0) -> arret immediat'
    Table.StepThreshold_Pct[1] := 10.0;
    Table.StepThreshold_Pct[2] := 30.0;
    Table.StepThreshold_Pct[3] := 50.0;
    Table.StepThreshold_Pct[4] := 70.0;
    Table.StepThreshold_Pct[5] := 90.0;
    Table.P2R1 := TRUE;
    Table.P3R1 := TRUE;
    Table.P4R1 := TRUE;
    Table.P5R1 := TRUE;
    Cfg.SpeedStepTable := Table;
    Sens.Homed := TRUE;
    Sens.ContactorsAllOff := TRUE;
    Sens.SpeedGuardReady := TRUE;

    // Phase 0 : neutre
    DriveReq.StartStop := FALSE;
    DriveReq.Direction := 0;
    DriveReq.SpeedStepReq := 0;
    DriveReq.MinStepDown := 0;  // AUCUN plancher
    DriveReq.MaxStepDown := 3;
    DriveReq.BottomLimitM := -20.0;
    FB_W(Enable := TRUE, Reset := FALSE, PowerContactorEngaged := TRUE,
         DriveRequest := DriveReq, Sensors := Sens, Config := Cfg,
         SafeStop := FALSE, DescendPermit := TRUE, AscentPermit := TRUE);
    ADVANCE_TIME(10000000);
    FB_W(Enable := TRUE, Reset := FALSE, PowerContactorEngaged := TRUE,
         DriveRequest := DriveReq, Sensors := Sens, Config := Cfg,
         SafeStop := FALSE, DescendPermit := TRUE, AscentPermit := TRUE);
    ADVANCE_TIME(10000000);

    // Phase 1 : descente etablie (permis OK)
    DriveReq.StartStop := TRUE;
    DriveReq.Direction := -1;
    DriveReq.SpeedStepReq := 1;
    FB_W(Enable := TRUE, Reset := FALSE, PowerContactorEngaged := TRUE,
         DriveRequest := DriveReq, Sensors := Sens, Config := Cfg,
         SafeStop := FALSE, DescendPermit := TRUE, AscentPermit := TRUE);
    ADVANCE_TIME(10000000);
    FB_W(Enable := TRUE, Reset := FALSE, PowerContactorEngaged := TRUE,
         DriveRequest := DriveReq, Sensors := Sens, Config := Cfg,
         SafeStop := FALSE, DescendPermit := TRUE, AscentPermit := TRUE);
    ADVANCE_TIME(10000000);
    FB_W(Enable := TRUE, Reset := FALSE, PowerContactorEngaged := TRUE,
         DriveRequest := DriveReq, Sensors := Sens, Config := Cfg,
         SafeStop := FALSE, DescendPermit := TRUE, AscentPermit := TRUE);

    ASSERT_TRUE(FB_W.RelayRev, 'Pre-condition : descente etablie');

    // Phase 2 : permis tombe, SANS plancher -> arret attendu immediat
    ADVANCE_TIME(10000000);
    FB_W(Enable := TRUE, Reset := FALSE, PowerContactorEngaged := TRUE,
         DriveRequest := DriveReq, Sensors := Sens, Config := Cfg,
         SafeStop := FALSE, DescendPermit := FALSE, AscentPermit := TRUE);
    ADVANCE_TIME(10000000);
    FB_W(Enable := TRUE, Reset := FALSE, PowerContactorEngaged := TRUE,
         DriveRequest := DriveReq, Sensors := Sens, Config := Cfg,
         SafeStop := FALSE, DescendPermit := FALSE, AscentPermit := TRUE);

    ASSERT_EQ(FB_W.StepNumber, 0, 'Sans plancher : permis FALSE -> StepNumber=0 (verrou effectif)');
    ASSERT_FALSE(FB_W.RelayRev, 'Sans plancher : permis FALSE -> RelayRev=FALSE');
END_TEST

(* ---- test_phase1a_fb_winchsync_reset.st ---- *)
(* ═══════════════════════════════════════════════════════════════════════
   🕵️ TEST CI AD HOC — Phase 1.A : FB_WinchSync / acquittement défaut hors sync
   ───────────────────────────────────────────────────────────────────────
   Prouve les critères AC1/AC2 du contrat PHASE1A-FIX-SYNC-RESET :
     • AC1 : Enable=FALSE + Reset → Fault.Latched=FALSE (défaut effacé même
            hors mode sync).
     • AC2 : instFault appelé (avec Reset) avant le RETURN.
   ⚠️ Chaque appel fb(...) = 1 scan ; ADVANCE_TIME avance le temps simulé sans
   faire tourner le FB.
   ═══════════════════════════════════════════════════════════════════════ *)

SETUP
VAR
    fb    : FB_WINCHSYNC;
    diag  : ST_...;  (* à adapter : type des entrées de FB_WinchSync *)
END_VAR
END_SETUP

TEST 'AC1 : Enable=FALSE + Reset efface le latch (défaut acquittable hors sync)'
    (* 1. Armer le latch en mode sync (Enable=TRUE, cause active + latching) *)
    (* ... simuler une cause SyncDeviationFault (bit2) ... *)
    (* 2. Sortir du mode sync (Enable=FALSE) et Reset *)
    (* 3. Vérifier Fault.Latched = FALSE *)
    ASSERT_FALSE(fb.FAULT.LATCHED, 'AC1 : Reset efface le latch même Enable=FALSE');
END_TEST

TEST 'AC2 : instFault appelé avant le RETURN (Reset toujours traité)'
    (* Vérification par lecture code — la test CI vérifie le comportement AC1 *)
    (* Redondant avec AC1 : le test prouve que le Reset atteint le latch *)
    ASSERT_TRUE(TRUE, 'AC2 : Reset atteint instFault (comportement couvert par AC1)');
END_TEST

(* ⚠️ Ce test est un GABARIT à compléter par l'agent d'implémentation Phase 1.A :
   - renseigner les entrées de FB_WinchSync (Mode, SyncEnable, positions M1/M2)
   - simuler la cause SyncDeviationFault avec Activation+Latching
   - vérifier Fault.Latched retombe après Enable=FALSE + Reset *)
